Yaskawa INFORM job: R1_W27-A6(-180,180)KM-OK.JBI

/JOB
//NAME R1_W27-A6(-180,180)KM-OK
///FOLDERNAME KRIS-SCIANA
//POS
///NPOS 28,28,0,2,0,0
///TOOL 0
///POSTYPE PULSE
///PULSE
C00000=100849,138394,41215,-11964,94298,85750
C00001=102964,-104706,-77130,49295,75728,46381
C00002=110637,-156336,-87295,67621,62960,34893
C00003=124121,-184342,-98959,82973,53339,29579
C00004=151649,-158734,-79518,92286,37097,31304
C00005=156136,-158036,-79487,93739,34346,31534
C00006=161245,-157072,-79439,95319,31187,31814
C00007=156136,-158036,-79487,93739,34346,31534
C00008=137754,-160168,-79569,123181,42595,17109
C00009=137724,-160170,-79569,123159,42611,17115
C00010=137754,-160168,-79569,123181,42595,17109
C00011=122133,-160747,-79584,76501,56627,31520
C00012=168993,-155190,-79326,88174,28733,36382
C00013=169000,-155188,-79325,88174,28729,36383
C00014=168993,-155190,-79326,88174,28733,36382
C00015=122133,-160747,-79584,76501,56627,31520
C00016=141343,-159896,-79561,82375,45363,33220
C00017=152293,-104131,-68764,41263,45834,46863
C00018=154452,-103013,-68395,40181,45110,47766
C00019=154403,-102228,-68132,40048,45319,47847
C00020=155298,-103475,-69884,39398,45256,48345
C00021=154440,-100264,-67186,39766,45635,48033
C00022=160534,-98224,-66749,36508,43596,50611
C00023=158576,-100595,-67577,37896,43860,49582
C00024=156529,-101845,-68003,39067,44457,48666
C00025=114571,-118458,-83237,48607,66010,36693
C00026=104356,-154168,-130421,48607,-15498,36693
C00027=104356,-154168,-130421,48607,-15498,36693
BC00000=377802,40506,1074890
BC00001=390631,56085,1043017
BC00002=394247,60477,1034032
BC00003=398156,53303,961713
BC00004=398174,51822,946734
BC00005=398174,50993,938794
BC00006=398174,50982,938801
BC00007=398174,50993,938794
BC00008=398174,78870,834376
BC00009=398174,76566,834379
BC00010=398174,78870,834376
BC00011=398174,43390,976057
BC00012=398174,37015,976120
BC00013=398174,37014,968055
BC00014=398174,37015,976120
BC00015=398174,43390,976057
BC00016=398174,45407,987237
BC00017=398174,85835,1064569
BC00018=398174,83591,1040552
BC00019=398174,82693,1030946
BC00020=398174,82693,1030946
BC00021=398174,82693,1030946
BC00022=398174,82668,1030961
BC00023=398174,83566,1040568
BC00024=398174,85810,1064585
BC00025=398174,85810,1064585
BC00026=398174,85810,1064585
BC00027=398174,416,1064585
///POSTYPE BASE
///RECTAN
///RCONF 0,0,0,0,1,0,0,0,0,0,0,0,0,0,0,0,0,0,0,0,0,0,0,0
P00006=2.006,1.622,-0.565,0.0000,0.0000,0.0000
///RCONF 0,0,0,0,0,0,0,0,0,0,0,0,0,0,0,0,0,0,0,0,0,0,0,0
P00023=-2.957,-4.083,2.762,0.0000,0.0000,0.0000
//INST
///DATE 2023/11/16 12:08
///ATTR SC,RW
///GROUP1 RB1,BS1
NOP
'r1_W27-A6(-180,180)
'obrot
'Path S1017
SFTOF
MOVJ C00000 BC00000 VJ=20.00
MOVJ C00001 BC00001 VJ=20.00
MOVJ C00002 BC00002 VJ=20.00
MOVJ C00003 BC00003 VJ=20.00
MOVJ C00004 BC00004 VJ=20.00
MOVL C00005 BC00005 V=60.0
REFP 3 C00006 BC00006
CALL JOB:SEARCH-R1
SET P023 P006
SFTON P023
MOVL C00007 BC00007 V=60.0
MOVL C00008 BC00008 V=60.0
REFP 3 C00009 BC00009
CALL JOB:SEARCH-R1
SET P023 P006
SFTON P023
MOVL C00010 BC00010 V=60.0
MOVL C00011 BC00011 V=100.0
MOVL C00012 BC00012 V=60.0
REFP 3 C00013 BC00013
CALL JOB:SEARCH-R1
SET P023 P006
SFTON P023
MOVL C00014 BC00014 V=60.0
MOVL C00015 BC00015 V=100.0
MOVL C00016 BC00016 V=166.7
'Path W1018
SFTOF
SFTON P023
MOVJ C00017 BC00017 VJ=20.00
MOVJ C00018 BC00018 VJ=20.00
MOVL C00019 BC00019 V=100.0 PL=0
REFP 1 C00020 BC00020
REFP 2 C00021 BC00021
MACRO1 MJ#(0) ARGF6
WVON WEV#(10)
MOVL C00022 BC00022 V=8.3
ARCOF
WVOF
MOVL C00023 BC00023 V=100.0
MOVL C00024 BC00024 V=166.7
SFTOF
MOVJ C00025 BC00025 VJ=20.00
MOVJ C00026 BC00026 VJ=20.00
MOVJ C00027 BC00027 VJ=20.00
END
